TYPE (* a Struct holding 2x3 Object IDs *)
  (* Version 1.0, 2026-05-28, Franz Höpfinger, Demmler Andreas Fahrzeugbau *)
  PACKAGE isobus::UT::Q::types;
  IMPORT isobus::UT::Q::const::IDs::ID_NULL;
  s2x3ObjectIDs : STRUCT
    up : isobus::UT::Q::types::s3ObjectIDs := (u16ObjId := ID_NULL, u16ObjIdA := ID_NULL, u16ObjIdB := ID_NULL); (* forward, up, right, clockwise *)
    down : isobus::UT::Q::types::s3ObjectIDs := (u16ObjId := ID_NULL, u16ObjIdA := ID_NULL, u16ObjIdB := ID_NULL); (* backward, down, left, counter-clockwise *)
  END_STRUCT;
END_TYPE
